Fanuc KAREL source: kc00035.KL

-- PROVISIONAL review KL for V770-1; original PC SHA256 a003b04211a707804468233cbccabe5328a9c82be803cfe683412dca4184bcab
-- Incomplete behavior may be omitted. Consult companion uncertainty JSON. Do not deploy.
PROGRAM KC00035
%NOLOCKGROUP
BEGIN
  -- UNRESOLVED_PC offsets 5-41; opcodes 27,22,22,2A,22,22,22,31
  -- UNRESOLVED_PC offsets 46-50; opcodes 7F
END KC00035
